PROGRAM SafetyConnect
VAR
END_VAR

IF GVL_HMI.MCR THEN
	IF GVL_Saf.InRun = 0 THEN
		GVL_Saf.Run := 0;
		GVL_Saf.ErrorAcknowledgment :=1;
	ELSE
		GVL_Saf.EStopReset := 1;
	END_IF	
ELSE
	GVL_Saf.EStopReset := 0;
	GVL_Saf.ErrorAcknowledgment :=0;
	GVL_Saf.Run := 1;
END_IF

END_PROGRAM

(* stored: Version 1.1.0.1, ProductVersion 3.1.4024.12
   POU SafetyConnect: Id {a2692ae3-b110-463e-a0c5-0930afb08b49}, SpecialFunc None *)
